SYSTEM System (* System Configuration *)
  (* Standard: 61499-1 *)
  (* Version 0.0, 14/06/2021, prana, Schneider Electric *)
  {SET_ATTRIBUTE(System.Device.FolderPath, DEV)}
  APPLICATION APP1
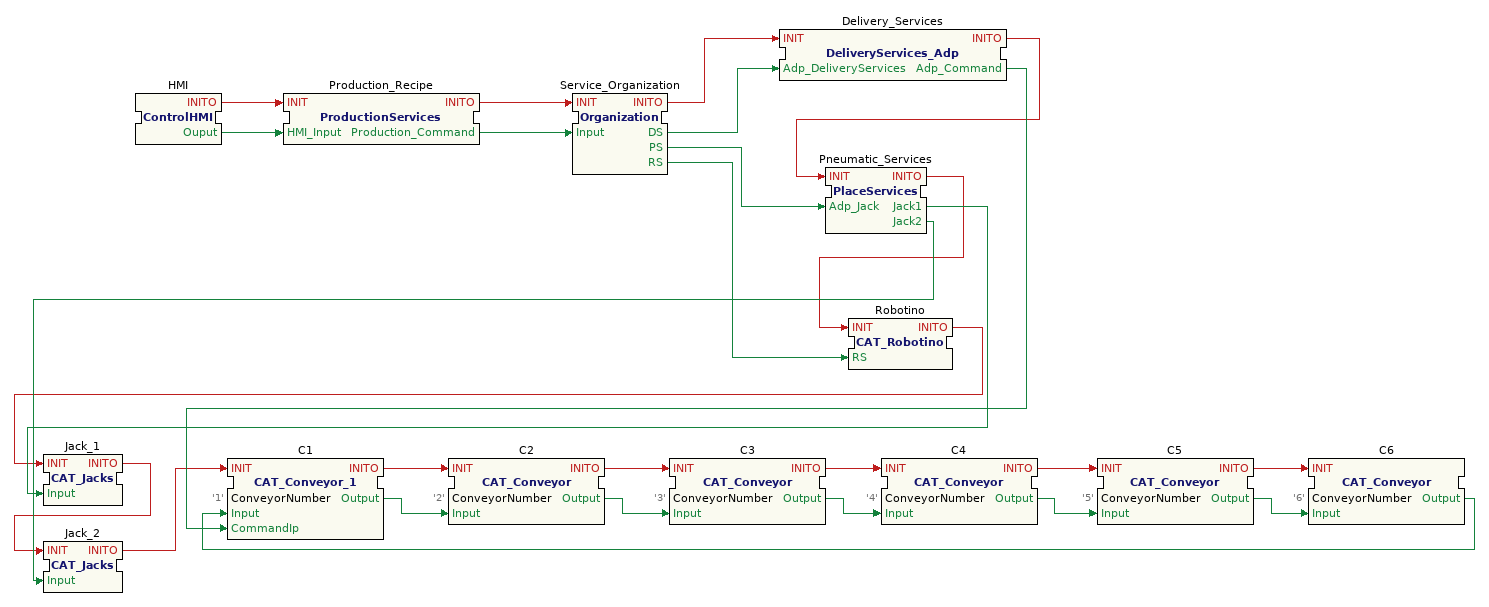
    (* Production Services *)
    (* Planning Services *)
    (* Order Services *)
    (* Execution Services *)
    FBS
      C4 : CAT_Conveyor(ConveyorNumber := '4');
      C2 : CAT_Conveyor(ConveyorNumber := '2');
      C1 : CAT_Conveyor_1(ConveyorNumber := '1');
      C3 : CAT_Conveyor(ConveyorNumber := '3');
      C5 : CAT_Conveyor(ConveyorNumber := '5');
      C6 : CAT_Conveyor(ConveyorNumber := '6');
      Delivery_Services : DeliveryServices_Adp;
      Production_Recipe : ProductionServices;
      Service_Organization : Organization;
      Pneumatic_Services : PlaceServices;
      Jack_1 : CAT_Jacks;
      Jack_2 : CAT_Jacks;
      HMI : ControlHMI;
      Robotino : CAT_Robotino;
    END_FBS
    EVENT_CONNECTIONS
      C1.INITO TO C2.INIT;
      C2.INITO TO C3.INIT;
      C3.INITO TO C4.INIT;
      C4.INITO TO C5.INIT;
      C5.INITO TO C6.INIT;
      Production_Recipe.INITO TO Service_Organization.INIT;
      Service_Organization.INITO TO Delivery_Services.INIT;
      Delivery_Services.INITO TO Pneumatic_Services.INIT;
      Pneumatic_Services.INITO TO Robotino.INIT;
      Jack_1.INITO TO Jack_2.INIT;
      Jack_2.INITO TO C1.INIT;
      HMI.INITO TO Production_Recipe.INIT;
      Robotino.INITO TO Jack_1.INIT;
    END_CONNECTIONS
    ADAPTER_CONNECTIONS
      C1.Output TO C2.Input;
      C2.Output TO C3.Input;
      C3.Output TO C4.Input;
      C4.Output TO C5.Input;
      C5.Output TO C6.Input;
      C6.Output TO C1.Input;
      Delivery_Services.Adp_Command TO C1.CommandIp;
      Production_Recipe.Production_Command TO Service_Organization.Input;
      Service_Organization.DS TO Delivery_Services.Adp_DeliveryServices;
      Service_Organization.PS TO Pneumatic_Services.Adp_Jack;
      Pneumatic_Services.Jack1 TO Jack_1.Input;
      Pneumatic_Services.Jack2 TO Jack_2.Input;
      HMI.Ouput TO Production_Recipe.HMI_Input;
      Service_Organization.RS TO Robotino.RS;
    END_CONNECTIONS
  END_APPLICATION
  DEVICE DEV : Soft_dPAC
    RESOURCE RES0 : EMB_RES_ECO
      FBS
        C1 : CAT_Conveyor_1(ConveyorNumber := '1');
        C2 : CAT_Conveyor(ConveyorNumber := '2');
        C3 : CAT_Conveyor(ConveyorNumber := '3');
        C4 : CAT_Conveyor(ConveyorNumber := '4');
        C5 : CAT_Conveyor(ConveyorNumber := '5');
        C6 : CAT_Conveyor(ConveyorNumber := '6');
        Delivery_Services : DeliveryServices_Adp;
        Production_Recipe : ProductionServices;
        Service_Organization : Organization;
        Pneumatic_Services : PlaceServices;
        Jack_1 : CAT_Jacks;
        Jack_2 : CAT_Jacks;
        HMI : ControlHMI;
        Robotino : CAT_Robotino;
      END_FBS
      EVENT_CONNECTIONS
        Delivery_Services.INITO TO Pneumatic_Services.INIT;
        Jack_1.INITO TO Jack_2.INIT;
        Jack_2.INITO TO C1.INIT;
        Pneumatic_Services.INITO TO Robotino.INIT;
        Robotino.INITO TO Jack_1.INIT;
        C1.INITO TO C2.INIT;
        C2.INITO TO C3.INIT;
        C3.INITO TO C4.INIT;
        C4.INITO TO C5.INIT;
        C5.INITO TO C6.INIT;
        START.COLD TO HMI.INIT;
        START.WARM TO HMI.INIT;
        Production_Recipe.INITO TO Service_Organization.INIT;
        Service_Organization.INITO TO Delivery_Services.INIT;
        HMI.INITO TO Production_Recipe.INIT;
      END_CONNECTIONS
      ADAPTER_CONNECTIONS
        C1.Output TO C2.Input;
        C2.Output TO C3.Input;
        C3.Output TO C4.Input;
        C4.Output TO C5.Input;
        C5.Output TO C6.Input;
        C6.Output TO C1.Input;
        Delivery_Services.Adp_Command TO C1.CommandIp;
        Production_Recipe.Production_Command TO Service_Organization.Input;
        Service_Organization.DS TO Delivery_Services.Adp_DeliveryServices;
        Service_Organization.PS TO Pneumatic_Services.Adp_Jack;
        Pneumatic_Services.Jack1 TO Jack_1.Input;
        Pneumatic_Services.Jack2 TO Jack_2.Input;
        HMI.Ouput TO Production_Recipe.HMI_Input;
        Service_Organization.RS TO Robotino.RS;
      END_CONNECTIONS
    END_RESOURCE
  END_DEVICE
  MAPPINGS
    APP1.C1 ON DEV.RES0;
    APP1.C2 ON DEV.RES0;
    APP1.C3 ON DEV.RES0;
    APP1.C4 ON DEV.RES0;
    APP1.C5 ON DEV.RES0;
    APP1.C6 ON DEV.RES0;
    APP1.Delivery_Services ON DEV.RES0;
    APP1.Production_Recipe ON DEV.RES0;
    APP1.Service_Organization ON DEV.RES0;
    APP1.Pneumatic_Services ON DEV.RES0;
    APP1.Jack_1 ON DEV.RES0;
    APP1.Jack_2 ON DEV.RES0;
    APP1.HMI ON DEV.RES0;
    APP1.Robotino ON DEV.RES0;
  END_MAPPINGS
END_SYSTEM
